TYPE T_ADC_CTRL EXTENDS T_MA_CTRL :
STRUCT
	lrTargetPos:    ARRAY [1..2] OF LREAL;
	lrTargetVel:    LREAL;
	lrPosang: 		ARRAY [1..2] OF LREAL;
END_STRUCT
END_TYPE

(* stored: Version 1.1.0.1, ProductVersion 3.1.4024.11
   DUT T_ADC_CTRL: Id {1ad5f44f-bffc-406b-801a-f8d493c0dacb} *)
